// TIA Portal V20 export
// export: Created 2025-09-12T17:14:00.0000000Z, ExportSetting WithDefaults, DisplayName Totally Integrated Automation Portal, DisplayVersion V20
FUNCTION_BLOCK "FB100_EM_SupplyFan"   // FB, SCL
TITLE = EM-100: Supply Fan Control
AUTHOR : Dallas Levine
VERSION : 0.1
// This block contains all logic for the Supply Fan Equipment Module (EM-100).
// stored: AutoNumber true, IsRetain false, StructureModified true
   VAR_INPUT
      Enable : Bool;   // Enables the block's execution.
   END_VAR
   VAR
      UDT : "UDT100_EM_SupplyFan";   // The data interface for the Supply Fan Equipment Module.
   END_VAR
BEGIN
// Initial network.
   REGION Placeholder for SCL Code 

   END_REGION
END_FUNCTION_BLOCK
